FUNCTION_BLOCK FB_axisCtrl
VAR_INPUT
	
END_VAR
VAR_OUTPUT
END_VAR
VAR_IN_OUT     
	stAxisCtrl	:ST_axisCtrl; 	
	IN_OUT 		: ST_MotionAxis_MC	;//struct for each axis
END_VAR
VAR

END_VAR

//add timeout for this fuction block
CASE stAxisCtrl.iCmd OF
	0:
		IN_OUT.mcReset.Execute	:= FALSE;
		IN_OUT.mcStop.Execute	:= FALSE	;
	1:
		IN_OUT.mcPower.Enable	:= TRUE;
		stAxisCtrl.iCmd	:= 0;
	2:
		IN_OUT.mcPower.Enable	:= FALSE;
		stAxisCtrl.iCmd	:= 0;	
	3:
		IN_OUT.mcReset.Execute	:= TRUE;
		stAxisCtrl.iCmd	:= 0;
	4:
		IN_OUT.mcStop.Execute	:= TRUE;
		stAxisCtrl.iCmd	:= 0;	
	5: 
		IN_OUT.mcMoveAbsolute.Execute := TRUE;
		IN_OUT.rActualPosSet	:= stAxisCtrl.rPosition;
		IN_OUT.rVelocitySet	:= stAxisCtrl.iSpeed;
		IF IN_OUT.mcMoveAbsolute.Done THEN
			stAxisCtrl.iCmd	:= 0;
		END_IF
END_CASE;
stAxisCtrl.iStatus := stAxisCtrl.iCmd;

END_FUNCTION_BLOCK

(* stored: Version 1.1.0.1, ProductVersion 3.1.4024.12
   POU FB_axisCtrl: Id {2ac385ec-b262-4b8e-ba8d-e1a3f0cb06b1}, SpecialFunc None *)
